// TIA Portal V17 export
// export: Created 2025-06-26T07:49:54.2451691Z, ExportSetting WithDefaults, DisplayName Totally Integrated Automation Portal, DisplayVersion V17 Update 8, DisplayName TIA Portal Openness, DisplayVersion V17 Update 8, DisplayName TIA Portal Version Control Interface, DisplayVersion V17, DisplayName STEP 7 Professional, DisplayVersion V17 Update 8, DisplayName STEP 7 Safety, DisplayVersion V17 Update 6, DisplayName WinCC Advanced, DisplayVersion V17 Update 8
TYPE "stET200AL_AQ"
// stored: IsFailsafeCompliant false
   STRUCT
      CH0 : Int;
      CH1 : Int;
      CH2 : Int;
      CH3 : Int;
      Spare : Byte;   // So AI & AQ have the same size
   END_STRUCT;
END_TYPE
